// TIA Portal V20 export
TYPE "typeCmControlNode"
// stored: Namespace Unit1.Em2
   STRUCT
      distanceOutPos : Bool;
      interlock : "Unit1.Em2.typeCmControlNodeInterlock";
      command : "Unit1.Em2.typeCmControlNodeCommand";
      softcam : "Unit1.Em2.typeCmControlNodeSoftCam";
      brakeTest : "Unit1.Em2.typeCmControlNodeBrakeTest";
      safeReferencing : "Unit1.Em2.typeCmHmiInterfaceSafeRef";
   END_STRUCT;
END_TYPE
